{attribute 'GeneratedUsingTerminal: EL3151-0000-0016'}
{attribute addProperty BoxType "EL3151-0000-0016"}
{attribute addProperty Description "EL3151 1Ch. Ana. Input 4-20mA"}
{attribute addProperty Physics "KK"}
{attribute addProperty Id "AI_StandardAT %I*AI_Standard_A8DF64E310WcStateAT %I*WcState_9091E0EB2InfoDataAT %I*InfoData_32EB74EA10"}
{attribute addProperty CRC "2916756744"}
{attribute addProperty Size "22"}
TYPE EL3151_ADDA2D08 EXTENDS EtcSlaveTerminalBase_947E5A46 :
STRUCT
	{attribute addProperty Name "AI_Standard"}
	AI_Standard : AI_Standard_A8DF64E3;
	{attribute addProperty Name "WcState"}
	WcState : WcState_9091E0EB;
	{attribute addProperty Name "InfoData"}
	InfoData : InfoData_32EB74EA;
END_STRUCT
END_TYPE

(* stored: Version 1.2.0.0, ProductVersion 3.1.4024.11
   DUT EL3151_ADDA2D08: Id {72efdd0d-2943-4e62-b932-76a7e33f69b6} *)
